// TwinCAT 3 PLC project LED_Sensors
// ProgramVersion: 3.1.4023.0
// libraries:
//   Tc2_ControllerToolbox, * (Beckhoff Automation GmbH)
//   Tc2_Standard, * (Beckhoff Automation GmbH)
//   Tc2_System, * (Beckhoff Automation GmbH)
//   Tc3_EventLogger, * (Beckhoff Automation GmbH)
//   Tc3_Module, * (Beckhoff Automation GmbH)
// project tree:
//   DUTs/ LEDColor.TcDUT, LEDMode.TcDUT
//   GVLs/ GVL.TcGVL
//   / PlcTask.TcTTO
//   POUs/ FB_BoxLED.TcPOU, FB_EventLogging.TcPOU, FB_RGBLED.TcPOU, MAIN.TcPOU
// real-time tasks:
//   TASK PlcTask: cycle T#1ms, priority 20, ADS port 350
// I/O:
//   DEVICE Gerät 1 (EtherCAT), AmsNetId 10.183.66.136.2.1
//     Klemme 1 (EK1100) [EK1100 EtherCAT-Koppler (2A E-Bus)]
//       Klemme 2 (EL2564) [EL2564 4 K. LED-Ausgang, 5...48 V DC, 4 A, RGBW]
//       Klemme 3 (EL9011) [EL9011 Endklemme]
// variable links:
//   LED Sensors/LED Sensors Instance <-> Device 1 (EtherCAT)/Term 1 (EK1100)/Term 2 (EL2564)
//     PlcTask Inputs/GVL.bRedError <-> PWM Inputs Channel 1/Status/Error
//     PlcTask Inputs/GVL.bRedWarning <-> PWM Inputs Channel 1/Status/Warning
//     PlcTask Outputs/GVL.iBlue <-> PWM Outputs Channel 3/PWM output
//     PlcTask Outputs/GVL.iGreen <-> PWM Outputs Channel 2/PWM output
//     PlcTask Outputs/GVL.iWhite <-> PWM Outputs Channel 1/PWM output

CONFIGURATION LED_Sensors
    RESOURCE PLC ON TwinCAT3
        TASK PlcTask(INTERVAL := T#1ms, PRIORITY := 20);
        PROGRAM MAIN WITH PlcTask : MAIN;
    END_RESOURCE
END_CONFIGURATION

// ---- DUTs/LEDColor.TcDUT
{attribute 'qualified_only'}
{attribute 'strict'}
{attribute 'to_string'}
TYPE LEDColor :
(
	Off,
	Red,
	Green,
	Blue
);
END_TYPE

// ---- DUTs/LEDMode.TcDUT
{attribute 'qualified_only'}
{attribute 'strict'}
{attribute 'to_string'}
TYPE LEDMode :
(
	Off,
	On,
	Dimmed,
	SlowFlashing,
	FastFlashing
);
END_TYPE

// ---- GVLs/GVL.TcGVL
{attribute 'qualified_only'}
VAR_GLOBAL
	iRed AT %Q* : INT;
	iGreen AT %Q* : INT;
	iBlue AT %Q* : INT;
	iWhite AT %Q* : INT;
	
	bRedWarning AT %I* : BOOL;
	bRedError AT %I* : BOOL;
END_VAR

// ---- POUs/MAIN.TcPOU
PROGRAM MAIN
VAR
	fbRGBLED : FB_RGBLED;
	fbBoxLED : FB_BoxLED;
	
	fbEventLogging : FB_EventLogging;
	
	eMode : LEDMode;
	eColor : LEDColor;
END_VAR

fbBoxLED.eMode := eMode;
fbRGBLED.eColor := eColor;

fbRGBLED();
fbBoxLED();

fbEventLogging();

END_PROGRAM

// ---- POUs/FB_RGBLED.TcPOU
FUNCTION_BLOCK FB_RGBLED
VAR_INPUT
	eColor : LEDColor;
END_VAR
VAR
	//Local
	iRedLED : INT;
	iGreenLED : INT;
	iBlueLED : INT;
	
	//ErrorBits
	bRedTemperatureTooHigh : BIT;
	bRedNoSupplyVoltage : BIT;
	bGreenTemperatureTooHigh : BIT;
	bGreenNoSupplyVoltage : BIT;
	bBlueTemperatureTooHigh : BIT;
	bBlueNoSupplyVoltage : BIT;	
END_VAR
VAR CONSTANT
	iMax : INT := 32767;		//Maximum Intensity (100%)
	iMin : INT := 0;			//Off (0%)
END_VAR

CASE eColor OF
	LEDColor.Off:
		iRedLED := iMin;
		iGreenLED := iMin;
		iBlueLED := iMin;
	LEDColor.Red:
		iRedLED := iMax;
		iGreenLED := iMin;
		iBlueLED := iMin;
	LEDColor.Green:
		iRedLED := iMin;
		iGreenLED := iMax;
		iBlueLED := iMin;
	LEDColor.Blue:
		iRedLED := iMin;
		iGreenLED := iMin;
		iBlueLED := iMax;
END_CASE

END_FUNCTION_BLOCK

// ---- POUs/FB_BoxLED.TcPOU
FUNCTION_BLOCK FB_BoxLED
VAR_INPUT
	eMode : LEDMode;
END_VAR
VAR
	//Local
	iBoxLED : INT;
	fbFlashingTimer : TON;
	bOn : BOOL;
	
	//ErrorBits
	bTemperatureTooHigh : BIT;
	bNoSupplyVoltage : BIT;
END_VAR
VAR CONSTANT
	iIntensity : INT := 32767;				//Intensity [0..32767]
	rDimFactor : REAL := 0.01;				//Percentage (0..100%)
	tSlowFlashingTime : TIME := T#1S;		
	tFastFlashingTime : TIME := T#100MS;
END_VAR

CASE eMode OF
	LEDMode.Off:
			doTurnOn(iBrightness := 0);
	LEDMode.On:
			doTurnOn(iBrightness := iIntensity);
	LEDMode.Dimmed:
			doDimming(rDimmingFactor:=rDimFactor);
	LEDMode.SlowFlashing:
			doFlashing(FlashingTime:=tSlowFlashingTime);
	LEDMode.FastFlashing:
			doFlashing(FlashingTime:=tFastFlashingTime);
END_CASE

METHOD PRIVATE doDimming
VAR_INPUT
	rDimmingFactor : REAL;
END_VAR
iBoxLED := REAL_TO_INT(rDimmingFactor * iIntensity);
END_METHOD

METHOD PRIVATE doFlashing
VAR_INPUT
	FlashingTime : TIME;
END_VAR
fbFlashingTimer(IN:=TRUE, PT:=FlashingTime);
IF fbFlashingTimer.Q THEN
	fbFlashingTimer(IN:=FALSE);
	bOn := NOT bOn;	
END_IF
IF bOn THEN
	iBoxLED := iIntensity;
ELSE
	iBoxLED := 0;
END_IF
END_METHOD

METHOD PRIVATE doTurnOn
VAR_INPUT
	iBrightness : INT;
END_VAR
iBoxLED := iBrightness;
END_METHOD

END_FUNCTION_BLOCK

// ---- POUs/FB_EventLogging.TcPOU
FUNCTION_BLOCK FB_EventLogging
VAR_INPUT
END_VAR
VAR_OUTPUT
END_VAR
VAR
	fbEventMessage : FB_TcMessage;
	fbEventLogger : FB_TcEventLogger;
	
	eMode : LEDMode;
	eColor : LEDColor;
	
	sColorAsString : STRING;
	sModeAsString : STRING;
	
	nCounter : UDINT;
END_VAR

sModeAsString := TO_STRING(MAIN.eMode);
IF eMode <> MAIN.eMode THEN
	eMode := MAIN.eMode; 
	fbEventMessage.CreateEx(stEventEntry:=TC_Events.LEDEvents.Mode, 0);
	fbEventMessage.ipArguments.AddString(sModeAsString);
	fbEventMessage.Send(0);
END_IF

sColorAsString := TO_STRING(MAIN.eColor);
IF eColor <> MAIN.eColor THEN
	eColor := MAIN.eColor; 
	fbEventMessage.CreateEx(stEventEntry:=TC_Events.LEDEvents.Color, 0);
	fbEventMessage.ipArguments.AddString(sColorAsString);
	fbEventMessage.Send(0);
END_IF

END_FUNCTION_BLOCK
